{attribute 'linkalways'} 
{attribute 'no_explicit_call' := 'This FB is a CLASS and must be accessed using methods or properties'}
{attribute 'enable_dynamic_creation'}
FUNCTION_BLOCK _ETcVnInterpolationType EXTENDS EnumDatatypeBase
VAR
	localData : ETcVnInterpolationType;
	activeData : REFERENCE TO ETcVnInterpolationType;
	enumBaseDatatype : _DINT(localData);
END_VAR

METHOD PRIVATE AddLocalEnumeration
VAR_INPUT
	Enumeration : T_MAXSTRING;
	Value : ETcVnInterpolationType;
END_VAR
AddEnumeration(Enumeration, Value);
END_METHOD

PROPERTY PUBLIC Address : PVOID
GET
Address := ADR(activeData);
END_GET
END_PROPERTY

METHOD PUBLIC ClearReference
VAR_INPUT
END_VAR
activeData REF= localData;
SetBaseDatatypeReference();
END_METHOD

METHOD PUBLIC Clone : I_Datatype
VAR
    pClone : POINTER TO _ETcVnInterpolationType;
END_VAR
pClone := __NEW(_ETcVnInterpolationType(InitialValue := Value));
Clone := pClone^;
END_METHOD

METHOD FB_init : BOOL
VAR_INPUT
	bInitRetains : BOOL; // if TRUE, the retain variables are initialized (warm start / cold start)
	bInCopyCode : BOOL;  // if TRUE, the instance afterwards gets moved into the copy code (online change)
	InitialValue : ETcVnInterpolationType;
END_VAR
localData := InitialValue;
AddBaseDatatype(enumBaseDatatype);
ClearReference();

AddLocalEnumeration('TCVN_IT_NEAREST_NEIGHBOR', ETcVnInterpolationType.TCVN_IT_NEAREST_NEIGHBOR);
AddLocalEnumeration('TCVN_IT_BILINEAR', ETcVnInterpolationType.TCVN_IT_BILINEAR);
AddLocalEnumeration('TCVN_IT_BICUBIC', ETcVnInterpolationType.TCVN_IT_BICUBIC);
AddLocalEnumeration('TCVN_IT_AREA_BASED', ETcVnInterpolationType.TCVN_IT_AREA_BASED);
AddLocalEnumeration('TCVN_IT_LANCZOS4', ETcVnInterpolationType.TCVN_IT_LANCZOS4);
END_METHOD

PROPERTY PUBLIC Identifier : T_MAXSTRING
GET
Identifier := 'ETcVnInterpolationType';
END_GET
END_PROPERTY

METHOD IsEnumeratorValueEqual : BOOL
VAR_INPUT
	Enumerator : I_KeyValueForwardEnumerator;
END_VAR
VAR
	storedValue : ETcVnInterpolationType;
END_VAR
IF NOT Enumerator.TryGet(storedValue) THEN
	RETURN;
END_IF

IsEnumeratorValueEqual := storedValue = activeData;
END_METHOD

METHOD PUBLIC MakeReferenceTo
VAR_INPUT
	ReferenceTarget : REFERENCE TO ETcVnInterpolationType;
END_VAR
activeData REF= ReferenceTarget;
SetBaseDatatypeReference();
END_METHOD

METHOD PROTECTED SetBaseDatatypeReference
VAR_INPUT
END_VAR
enumBaseDatatype.MakeReferenceTo(activeData);
END_METHOD

PROPERTY PUBLIC Size : UDINT
GET
Size := SIZEOF(activeData);
END_GET
END_PROPERTY

METHOD TryMakeReferenceTo : BOOL
VAR_INPUT
	Target : I_Datatype;
END_VAR
VAR
	targetAsEnum : I_EnumDatatype;
	pTargetData : POINTER TO ETcVnInterpolationType;
END_VAR
IF NOT Target.TryResolveAsEnumDatatype(targetAsEnum) THEN
	RETURN;
END_IF

IF targetAsEnum.Identifier <> Identifier THEN
	RETURN;
END_IF

pTargetData := Target.Address;
activeData REF= pTargetData^;
SetBaseDatatypeReference();
TryMakeReferenceTo := TRUE;
END_METHOD

PROPERTY PUBLIC Value : ETcVnInterpolationType
GET
Value := activeData;
END_GET
SET
activeData := Value;
END_SET
END_PROPERTY

END_FUNCTION_BLOCK

(* stored: Version 1.1.0.1, ProductVersion 3.1.4024.12
   POU _ETcVnInterpolationType: Id {ba9e75ea-42dd-0bba-233c-e8fdd72b7315}, SpecialFunc None
   Folder Constructor: Id {a2ff181c-f51e-0479-348a-e32c0d30ae23}
   Folder Private: Id {961f7734-5d31-09b1-3480-324fad025a32}
   Folder Protected: Id {bf471ec0-62d3-0704-05f2-765715c5bf74}
   Method AddLocalEnumeration: Id {c52ca102-bfe5-07b9-1f0f-1b385daa1fec}
   Property Address: Id {72bc1fed-4afd-0f22-3fb0-b7e22dc68dbf}
   Get Get: Id {d7f4a774-9065-07e0-0d3b-25048937d6bf}
   Method ClearReference: Id {37479d16-706c-031d-3183-71d77836d17b}
   Method Clone: Id {3c68b57b-e257-0887-0db6-d00ba9f9a5c2}
   Method FB_init: Id {90e6fcdb-3b53-0644-35b4-51f2e1bb969c}
   Property Identifier: Id {c2ac3934-f58a-015c-19a8-f155e14a13da}
   Get Get: Id {39b3ba09-cd88-08a5-050f-0a240e2f6694}
   Method IsEnumeratorValueEqual: Id {19d17fe2-2b7d-0e09-3445-a3de39075fe9}
   Method MakeReferenceTo: Id {5a39876c-d73c-0800-074d-07a171eca940}
   Method SetBaseDatatypeReference: Id {e7fb5f70-de95-01b7-176c-207c2725e913}
   Property Size: Id {ff2b9eb2-4108-0ae6-2caf-2b50dc886e1c}
   Get Get: Id {4ca2f391-a4ae-0b40-220a-811afe739000}
   Method TryMakeReferenceTo: Id {0070a147-d899-0157-3023-ed6c565d9c8a}
   Property Value: Id {662a6ce0-39e8-0e0d-2616-1e054740c6bd}
   Get Get: Id {121c3126-750d-02b1-02c6-0edc3f72b472}
   Set Set: Id {bf453bde-a1bb-025e-3b7d-10af8115e3d8} *)
